Fanuc KAREL source: kb00011.KL

-- PROVISIONAL review KL for V940-1; original PC SHA256 3cdeee3366deccf5371e60067222938ad1197aca563b1265fd9923d088b634eb
-- Incomplete behavior may be omitted. Consult companion uncertainty JSON. Do not deploy.
PROGRAM KB00011
%NOLOCKGROUP
BEGIN
  -- V9_ZERO_TABLE_METADATA_HINT layout=0002_ascii; no indexed target words; source/name/runtime held
  -- UNRESOLVED_PC offsets 5-14; opcodes 3F,75
  -- UNRESOLVED_PC offsets 19-28; opcodes 3F,75
  -- UNRESOLVED_PC offsets 33-40; opcodes 9D,23
  -- UNRESOLVED_PC offsets 45-52; opcodes 9D,23
  -- UNRESOLVED_PC offsets 57-64; opcodes 9D,23
  -- UNRESOLVED_PC offsets 69-107; opcodes 27,22,2A,22,2A,22,22,22,31
  -- UNRESOLVED_PC offsets 112-116; opcodes 7F
END KB00011
